FUNCTION_BLOCK CONTROL_PLANES
  (* Standard: 61499-2 *)
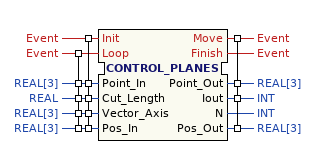
  EVENT_INPUT
    Init WITH Point_In, Cut_Length, Vector_Axis, Pos_In;
    Loop WITH Point_In, Cut_Length, Vector_Axis, Pos_In;
  END_EVENT
  EVENT_OUTPUT
    Move WITH Point_Out, Iout, Pos_Out;
    Finish;
  END_EVENT
  VAR_INPUT
    Point_In : ARRAY [0..2] OF REAL;
    Cut_Length : REAL;
    Vector_Axis : ARRAY [0..2] OF REAL;
    Pos_In : ARRAY [0..2] OF REAL;
  END_VAR
  VAR_OUTPUT
    Point_Out : ARRAY [0..2] OF REAL;
    Iout : INT;
    N : INT;
    Pos_Out : ARRAY [0..2] OF REAL;
  END_VAR
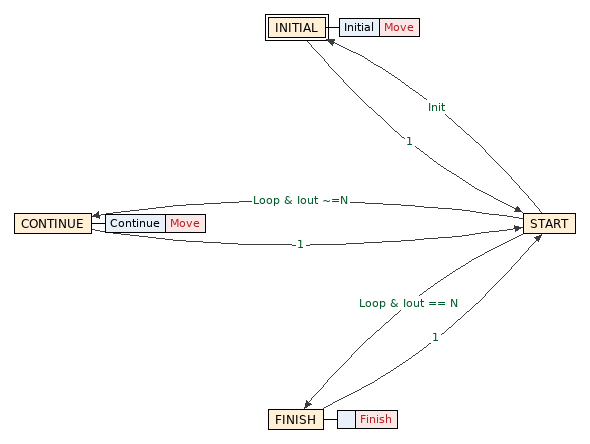
  EC_STATES
    INITIAL : Initial -> Move;
    START;
    FINISH : -> Finish;
    CONTINUE : Continue -> Move;
  END_STATES
  EC_TRANSITIONS
    START TO INITIAL := Init;
    START TO CONTINUE := Loop & Iout ~=N;
    START TO FINISH := Loop & Iout == N;
    FINISH TO START := 1;
    INITIAL TO START := 1;
    CONTINUE TO START := 1;
  END_TRANSITIONS
  ALGORITHM Initial IN Lua:
 N = -Point_In[3]/Cut_Length N = ceil(N) print( '\nN', N, Point_In[3], Cut_Length, '\n' ) if N==0 then N=1 end if Vector_Axis == '$' or not Vector_Axis or (Vector_Axis[1] == 0 and Vector_Axis[2] == 0 and Vector_Axis[3] ==0 ) then  Vector_Axis = {0, 0, 1} end   local an       = {0,0,1} Iout     = 1 Point_Out[3] = Point_In[3]/N local deltaz = (-1 + 1/N)*Point_In[3] local r      = deltaz/an[3] Point_Out[1] = Point_In[1] + r*an[1] Point_Out[2] = Point_In[2] + r*an[2]   local dz = Point_Out[3] local r2 = dz/an[3] local dx = r2*an[1] local dy = r2*an[2]   Pos_Out = {Pos_In[1] , Pos_In[2] , Pos_In[3] + deltaz} print('CONTROL PLANES Pos_Out', Pos_In[1] , Pos_In[2] , Pos_In[3] + deltaz) --local an = Vector_Axis local m  = sqrt(an[1]^2 + an[2]^2 + an[3]^2)
  END_ALGORITHM
  ALGORITHM Continue IN Lua:
 local an  = {0, 0, 1} Iout = Iout+1 Point_Out[3] = Point_In[3]*Iout/N local deltaz = (-1 + Iout/(N) )*Point_In[3] local r = deltaz/an[3] Point_Out[1] = Point_In[1] Point_Out[2] = Point_In[2]  local dz = Point_Out[3] - Point_In[3] local r2 = dz/an[3] local dx = r2*an[1] local dy = r2*an[2]  Pos_Out = {Pos_In[1] , Pos_In[2] , Pos_In[3] + dz} print('CONTROL PLANES Pos Out', Pos_In[1] + dx, Pos_In[2] + dy, Pos_In[3] + dz)
  END_ALGORITHM
END_FUNCTION_BLOCK
